Universal Robots PolyScope program: _adminCG-AssembleCLidToD.urp

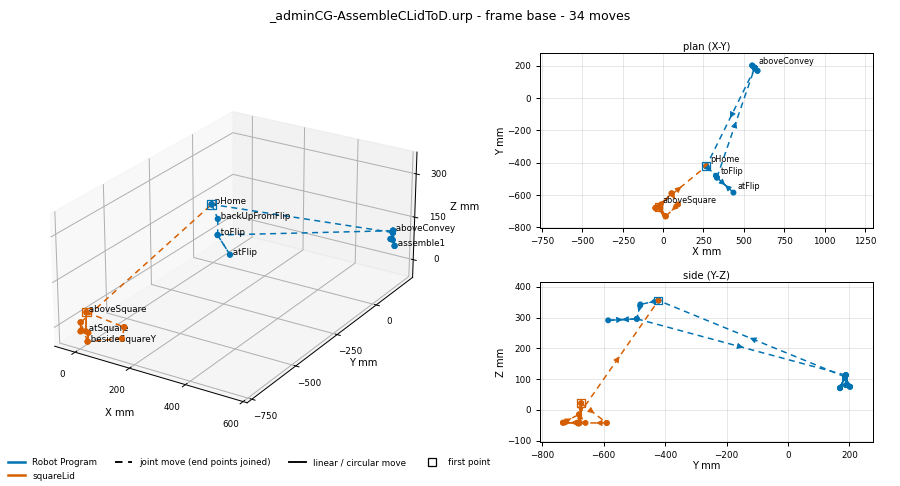
[picture p0: tool path of _adminCG-AssembleCLidToD.urp in frame base, 34 of 35 moves have a stored position in this frame; points joined in program order, loops and branches not executed]
Program _adminCG-AssembleCLidToD (installation=admin directory=/programs/WED_9AM createdIn=3.15.8.106339 lastSavedIn=3.15.8.106339 robotSerialNumber=2015350924)
Calibrated DH parameters: a=[0, -0.425, -0.39225, 0, 0, 0]; d=[0.089159, 0, 0, 0.10915, 0.09465, 0.0823]; alpha=[1.570796, 0, 0, 1.570796, -1.570796, 0]; deltaTheta=[0, 0, 0, 0, 0, 0]
Robot Program (runOnlyOnce=true)
  Set DigitalOutput pin=digital_out[0]; digitalValue=0
  MoveJ speed 60 deg/s, acceleration 80 deg/s^2 (useActiveTCP=true)
    Waypoint pHome: TCP in base x=267.157 y=-421.439 z=355.893 mm, rx=1.1139 ry=1.106 rz=0.0052 rad; joints [-44.996, -89.999, -89.997, -90.001, 90.007, 0.005] deg; flange x=267.148 y=-421.443 z=431.893 mm, rx=-1.2022 ry=2.9023 rz=0 rad
    Waypoint backUpFromFlip: TCP in base x=326.754 y=-480.276 z=343.158 mm, rx=1.1302 ry=1.1244 rz=-0.0012 rad; joints [-44.863, -101.867, -78.33, -91.204, 89.722, 0.314] deg; flange x=328.332 y=-481.325 z=419.134 mm, rx=1.1925 ry=-2.8912 rz=-0.0323 rad
  MoveJ speed 60 deg/s, acceleration 80 deg/s^2 (useActiveTCP=true)
    Call _adminLinearIndex4
    Waypoint toFlip: TCP in base x=333.102 y=-491.704 z=296.298 mm, rx=-1.5769 ry=1.6129 rz=-2.1772 rad; joints [-45.149, -123.398, -107.093, -41.475, -89.463, -0.24] deg; flange x=331.768 y=-489.353 z=220.346 mm, rx=0.0362 ry=0.0046 rz=0.7784 rad
    Waypoint atFlip: TCP in base x=435.484 y=-584.937 z=291.512 mm, rx=1.5199 ry=-1.5359 rz=2.2678 rad; joints [-44.833, -139.316, -77.941, -49.924, -90.495, -0.843] deg; flange x=437.672 y=-588.039 z=215.607 mm, rx=-0.0499 ry=-0.0116 rz=0.7732 rad
    Set DigitalOutput pin=digital_out[0]; digitalValue=1
    Wait Sleep waitTime=1
    Set DigitalOutput pin=digital_out[2]; digitalValue=0
    Wait Sleep waitTime=1
    Waypoint toFlip: TCP in base x=333.102 y=-491.704 z=296.298 mm, rx=-1.5769 ry=1.6129 rz=-2.1772 rad; joints [-45.149, -123.398, -107.093, -41.475, -89.463, -0.24] deg; flange x=331.768 y=-489.353 z=220.346 mm, rx=0.0362 ry=0.0046 rz=0.7784 rad
    Call _adminLinearIndex2
    Call squareLid
  MoveJ speed 60 deg/s, acceleration 80 deg/s^2 (useActiveTCP=true)
    Call _adminLinearIndex1
    Waypoint aboveConvey: TCP in base x=567.181 y=188.05 z=113.063 mm, rx=1.0282 ry=1.0751 rz=-0.0229 rad; joints [30.268, -112.359, -99.942, -58.865, 84.81, 74.946] deg; flange x=565.046 y=194.763 z=188.736 mm, rx=1.2073 ry=-2.8879 rz=0.1448 rad
    Waypoint rotateAbove: TCP in base x=567.194 y=188.064 z=113.07 mm, rx=1.5788 ry=-1.6466 rz=-2.1023 rad; joints [30.269, -112.36, -99.938, -58.868, 84.807, 254.946] deg; flange x=565.057 y=194.781 z=188.743 mm, rx=2.8131 ry=1.1761 rz=-0.0125 rad
    Waypoint atBody: TCP in base x=567.179 y=188.066 z=80.552 mm, rx=1.5785 ry=-1.6465 rz=-2.1025 rad; joints [30.268, -114.89, -101.837, -54.448, 84.816, 254.947] deg; flange x=565.059 y=194.78 z=156.225 mm, rx=2.8132 ry=1.1761 rz=-0.0127 rad
    Wait Sleep waitTime=1
    Set DigitalOutput pin=digital_out[0]; digitalValue=0
    Wait Sleep waitTime=1
    Waypoint rotateAbove: TCP in base x=567.194 y=188.064 z=113.07 mm, rx=1.5788 ry=-1.6466 rz=-2.1023 rad; joints [30.269, -112.36, -99.938, -58.868, 84.807, 254.946] deg; flange x=565.057 y=194.781 z=188.743 mm, rx=2.8131 ry=1.1761 rz=-0.0125 rad
    Waypoint aboveConvey: TCP in base x=567.181 y=188.05 z=113.063 mm, rx=1.0282 ry=1.0751 rz=-0.0229 rad; joints [30.268, -112.359, -99.942, -58.865, 84.81, 74.946] deg; flange x=565.046 y=194.763 z=188.736 mm, rx=1.2073 ry=-2.8879 rz=0.1448 rad
    Set DigitalOutput pin=digital_out[0]; digitalValue=1
    Waypoint abovePress: TCP in base x=568.039 y=185.31 z=107.717 mm, rx=1.0319 ry=1.117 rz=-0.0467 rad; joints [29.644, -113.286, -98.834, -61.278, 86.104, 74.264] deg; flange x=569.391 y=192.021 z=183.408 mm, rx=1.1944 ry=-2.8486 rz=0.1154 rad
  If force()≤65 (checkContinuously=true)
    MoveL speed 50 mm/s, acceleration 100 mm/s^2 (useActiveTCP=true) feature=Base
      Waypoint assemble1: TCP in base x=584.239 y=169.152 z=70.781 mm, rx=1.0609 ry=1.0742 rz=-0.0387 rad; joints [27.519, -116.934, -100.349, -53.785, 86.094, 73.63] deg; flange x=583.102 y=174.396 z=146.592 mm, rx=1.1698 ry=-2.9008 rz=0.109 rad
  MoveJ speed 60 deg/s, acceleration 80 deg/s^2 (useActiveTCP=true)
    Waypoint abovePress: TCP in base x=568.039 y=185.31 z=107.717 mm, rx=1.0319 ry=1.117 rz=-0.0467 rad; joints [29.644, -113.286, -98.834, -61.278, 86.104, 74.264] deg; flange x=569.391 y=192.021 z=183.408 mm, rx=1.1944 ry=-2.8486 rz=0.1154 rad
  If force()≤65 (checkContinuously=true)
    MoveL speed 50 mm/s, acceleration 100 mm/s^2 (useActiveTCP=true) feature=Base
      Waypoint assemble2: TCP in base x=551.811 y=201.79 z=75.225 mm, rx=1.0098 ry=1.1381 rz=-0.0159 rad; joints [31.851, -114.685, -102.439, -56.33, 86.144, 74.216] deg; flange x=552.994 y=208.542 z=150.915 mm, rx=1.2503 ry=-2.8248 rz=0.116 rad
  MoveJ speed 60 deg/s, acceleration 80 deg/s^2 (useActiveTCP=true)
    Waypoint abovePress: TCP in base x=568.039 y=185.31 z=107.717 mm, rx=1.0319 ry=1.117 rz=-0.0467 rad; joints [29.644, -113.286, -98.834, -61.278, 86.104, 74.264] deg; flange x=569.391 y=192.021 z=183.408 mm, rx=1.1944 ry=-2.8486 rz=0.1154 rad
  If force()≤65 (checkContinuously=true)
    MoveL speed 50 mm/s, acceleration 100 mm/s^2 (useActiveTCP=true) feature=Base
      Waypoint assemble1: TCP in base x=584.239 y=169.152 z=70.781 mm, rx=1.0609 ry=1.0742 rz=-0.0387 rad; joints [27.519, -116.934, -100.349, -53.785, 86.094, 73.63] deg; flange x=583.102 y=174.396 z=146.592 mm, rx=1.1698 ry=-2.9008 rz=0.109 rad
  MoveJ speed 60 deg/s, acceleration 80 deg/s^2 (useActiveTCP=true)
    Waypoint abovePress: TCP in base x=568.039 y=185.31 z=107.717 mm, rx=1.0319 ry=1.117 rz=-0.0467 rad; joints [29.644, -113.286, -98.834, -61.278, 86.104, 74.264] deg; flange x=569.391 y=192.021 z=183.408 mm, rx=1.1944 ry=-2.8486 rz=0.1154 rad
  If force()≤65 (checkContinuously=true)
    MoveL speed 50 mm/s, acceleration 100 mm/s^2 (useActiveTCP=true) feature=Base
      Waypoint assemble2: TCP in base x=551.811 y=201.79 z=75.225 mm, rx=1.0098 ry=1.1381 rz=-0.0159 rad; joints [31.851, -114.685, -102.439, -56.33, 86.144, 74.216] deg; flange x=552.994 y=208.542 z=150.915 mm, rx=1.2503 ry=-2.8248 rz=0.116 rad
  MoveJ speed 60 deg/s, acceleration 80 deg/s^2 (useActiveTCP=true)
    Waypoint abovePress: TCP in base x=568.039 y=185.31 z=107.717 mm, rx=1.0319 ry=1.117 rz=-0.0467 rad; joints [29.644, -113.286, -98.834, -61.278, 86.104, 74.264] deg; flange x=569.391 y=192.021 z=183.408 mm, rx=1.1944 ry=-2.8486 rz=0.1154 rad
    Waypoint pHome: TCP in base x=267.157 y=-421.439 z=355.893 mm, rx=1.1139 ry=1.106 rz=0.0052 rad; joints [-44.996, -89.999, -89.997, -90.001, 90.007, 0.005] deg; flange x=267.148 y=-421.443 z=431.893 mm, rx=-1.2022 ry=2.9023 rz=0 rad
SubProgram -> _adminLinearIndex1
SubProgram -> _adminLinearIndex4
SubProgram -> squareLid
SubProgram _adminLinearIndex3 (keepSynchronizedWithDisk=false) programFile=/programs/me345_admin/_adminLinearIndex3.urp
  Folder Move_linear_slide_Index1
    var_1 := False
    Loop While (checkContinuously=false) expression=var_1≟ False
      var_1 := socket_open("10.241.34.52",4001)
    var_3 := 1
    Send := "s r0x24 21"
    Script: socket_send_string(Send)
    Script: socket_send_byte(13)
    Send_Reply := socket_read_string()
    Send := "s r0xca 103936"
    Script: socket_send_string(Send)
    Script: socket_send_byte(13)
    Send_Reply := socket_read_string()
    Send := "t 1"
    Script: socket_send_string(Send)
    Script: socket_send_byte(13)
    Send_Reply := socket_read_string()
    Loop While (checkContinuously=false) expression=var_3≠0
      Send := "g r0xA0"
      Script: socket_send_string(Send)
      Script: socket_send_byte(13)
      var_3 := socket_get_var("v")
      Wait Sleep waitTime=0.1
    Script: socket_close()
    Script: sync()
SubProgram -> _adminLinearIndex2
SubProgram _adminLinearIndex5 (keepSynchronizedWithDisk=false) programFile=/programs/me345_admin/_adminLinearIndex5.urp
  Folder Move_linear_slide_Index5
    var_1 := False
    Loop While (checkContinuously=false) expression=var_1≟ False
      var_1 := socket_open("10.241.34.52",4001)
    var_3 := 1
    Send := "s r0x24 21"
    Script: socket_send_string(Send)
    Script: socket_send_byte(13)
    Send_Reply := socket_read_string()
    Send := "s r0xca 190000"
    Script: socket_send_string(Send)
    Script: socket_send_byte(13)
    Send_Reply := socket_read_string()
    Send := "t 1"
    Script: socket_send_string(Send)
    Script: socket_send_byte(13)
    Send_Reply := socket_read_string()
    Loop While (checkContinuously=false) expression=var_3≠0
      Send := "g r0xA0"
      Script: socket_send_string(Send)
      Script: socket_send_byte(13)
      var_3 := socket_get_var("v")
      Wait Sleep waitTime=0.1
    Script: socket_close()
    Script: sync()
SubProgram _adminLinearIndex4 (keepSynchronizedWithDisk=false) programFile=/programs/me345_admin/_adminLinearIndex4.urp
  Folder Move_linear_slide_Index4
    var_1 := False
    Loop While (checkContinuously=false) expression=var_1≟ False
      var_1 := socket_open("10.241.34.52",4001)
    var_3 := 1
    Send := "s r0x24 21"
    Script: socket_send_string(Send)
    Script: socket_send_byte(13)
    Send_Reply := socket_read_string()
    Send := "s r0xca 169167"
    Script: socket_send_string(Send)
    Script: socket_send_byte(13)
    Send_Reply := socket_read_string()
    Send := "t 1"
    Script: socket_send_string(Send)
    Script: socket_send_byte(13)
    Send_Reply := socket_read_string()
    Loop While (checkContinuously=false) expression=var_3≠0
      Send := "g r0xA0"
      Script: socket_send_string(Send)
      Script: socket_send_byte(13)
      var_3 := socket_get_var("v")
      Wait Sleep waitTime=0.1
    Script: socket_close()
    Script: sync()
SubProgram _adminLinearIndex2 (keepSynchronizedWithDisk=false) programFile=/programs/me345_admin/_adminLinearIndex2.urp
  Folder Move_linear_slide_Index2
    var_1 := False
    Loop While (checkContinuously=false) expression=var_1≟ False
      var_1 := socket_open("10.241.34.52",4001)
    var_3 := 1
    Send := "s r0x24 21"
    Script: socket_send_string(Send)
    Script: socket_send_byte(13)
    Send_Reply := socket_read_string()
    Send := "s r0xca 51968"
    Script: socket_send_string(Send)
    Script: socket_send_byte(13)
    Send_Reply := socket_read_string()
    Send := "t 1"
    Script: socket_send_string(Send)
    Script: socket_send_byte(13)
    Send_Reply := socket_read_string()
    Loop While (checkContinuously=false) expression=var_3≠0
      Send := "g r0xA0"
      Script: socket_send_string(Send)
      Script: socket_send_byte(13)
      var_3 := socket_get_var("v")
      Wait Sleep waitTime=0.1
    Script: socket_close()
    Script: sync()
SubProgram squareLid (keepSynchronizedWithDisk=false) programFile=/programs/WED_9AM/squareLid.urp
  MoveJ speed 180 deg/s, acceleration 100 deg/s^2 (useActiveTCP=true)
    Waypoint aboveSquare: TCP in base x=-28.511 y=-672.755 z=21.747 mm, rx=1.7065 ry=-0.0121 rz=-1.2064 rad; joints [-83.109, -128.084, -90.371, -51.361, 90.044, 52.13] deg; flange x=-28.598 y=-672.52 z=97.746 mm, rx=1.2074 ry=2.8979 rz=-0.0038 rad
  MoveL speed 250 mm/s, acceleration 1200 mm/s^2 (useActiveTCP=true) feature=Base
    Waypoint atSquare: TCP in base x=-30.006 y=-677.246 z=-41.376 mm, rx=1.7064 ry=-0.0122 rz=-1.2062 rad; joints [-83.283, -134.212, -90.751, -44.844, 90.048, 51.953] deg; flange x=-30.099 y=-676.998 z=34.624 mm, rx=1.2073 ry=2.8978 rz=-0.004 rad
    Set DigitalOutput pin=digital_out[0]; digitalValue=0
    Wait Sleep waitTime=0.5
    Waypoint aboveSquare: TCP in base x=-28.511 y=-672.755 z=21.747 mm, rx=1.7065 ry=-0.0121 rz=-1.2064 rad; joints [-83.109, -128.084, -90.371, -51.361, 90.044, 52.13] deg; flange x=-28.598 y=-672.52 z=97.746 mm, rx=1.2074 ry=2.8979 rz=-0.0038 rad
    Set DigitalOutput pin=digital_out[0]; digitalValue=1
  MoveJ speed 60 deg/s, acceleration 80 deg/s^2 (useActiveTCP=true)
    Waypoint besideSquareX: TCP in base x=52.617 y=-589.571 z=-42.423 mm, rx=1.7065 ry=-0.0117 rz=-1.2076 rad; joints [-74.267, -126.531, -106.897, -36.426, 89.974, 61.001] deg; flange x=52.598 y=-589.375 z=33.577 mm, rx=1.2085 ry=2.8985 rz=-0.0036 rad
  MoveL speed 35 mm/s, acceleration 35 mm/s^2 (useActiveTCP=true) feature=Base
    If force()≤40 (checkContinuously=true)
      Waypoint atSquareX_1 (Relative): relativeFromPosition TCP in base x=50.865 y=-591.008 z=-41.515 mm, rx=1.7022 ry=-0.008 rz=-1.2089 rad; joints [-74.266, -126.532, -106.898, -36.426, 89.971, 60.977] deg; TCP in base x=-28.314 y=-672.475 z=-41.562 mm, rx=1.7067 ry=-0.0121 rz=-1.2064 rad; joints [-83.089, -133.766, -91.707, -44.351, 90.046, 52.151] deg; flange x=-28.404 y=-672.249 z=34.438 mm, rx=1.2075 ry=2.8979 rz=-0.0036 rad
    Wait Sleep waitTime=0.5
  MoveJ speed 60 deg/s, acceleration 80 deg/s^2 (useActiveTCP=true)
    Waypoint besideSquareX: TCP in base x=52.617 y=-589.571 z=-42.423 mm, rx=1.7065 ry=-0.0117 rz=-1.2076 rad; joints [-74.267, -126.531, -106.897, -36.426, 89.974, 61.001] deg; flange x=52.598 y=-589.375 z=33.577 mm, rx=1.2085 ry=2.8985 rz=-0.0036 rad
    Waypoint linkingMove: motionParameters(blendRadius=0.01); TCP in base x=92.406 y=-658.703 z=-42.29 mm, rx=1.7071 ry=-0.0114 rz=-1.2067 rad; joints [-72.572, -133.085, -93.255, -43.522, 90.01, 62.663] deg; flange x=92.339 y=-658.532 z=33.709 mm, rx=1.2075 ry=2.8984 rz=-0.0027 rad
    Waypoint besideSquareY: TCP in base x=16.11 y=-732.019 z=-41.564 mm, rx=1.7069 ry=-0.0118 rz=-1.2058 rad; joints [-80.178, -139.758, -79.322, -50.745, 90.056, 55.034] deg; flange x=15.998 y=-731.803 z=34.435 mm, rx=1.2067 ry=2.8979 rz=-0.0032 rad
  MoveL speed 35 mm/s, acceleration 35 mm/s^2 (useActiveTCP=true) feature=Base
    If force()≤40 (checkContinuously=true)
      Waypoint atSquareY_1: TCP in base x=-16.892 y=-681.869 z=-41.456 mm, rx=1.7062 ry=-0.0123 rz=-1.2065 rad; joints [-82.218, -134.623, -89.92, -45.26, 90.031, 53.025] deg; flange x=-16.969 y=-681.614 z=34.543 mm, rx=1.2075 ry=2.8978 rz=-0.0043 rad
    Wait Sleep waitTime=0.5
  MoveJ speed 60 deg/s, acceleration 80 deg/s^2 (useActiveTCP=true)
    Waypoint besideSquareY: TCP in base x=16.11 y=-732.019 z=-41.564 mm, rx=1.7069 ry=-0.0118 rz=-1.2058 rad; joints [-80.178, -139.758, -79.322, -50.745, 90.056, 55.034] deg; flange x=15.998 y=-731.803 z=34.435 mm, rx=1.2067 ry=2.8979 rz=-0.0032 rad
    Waypoint aboveSquareNew: TCP in base x=-46.625 y=-679.478 z=-14.514 mm, rx=1.7065 ry=-0.012 rz=-1.2064 rad; joints [-84.714, -132.04, -89.733, -48.043, 90.045, 50.52] deg; flange x=-46.706 y=-679.241 z=61.486 mm, rx=1.2073 ry=2.898 rz=-0.0039 rad
    Set DigitalOutput pin=digital_out[0]; digitalValue=0
    Wait Sleep waitTime=1
  MoveL speed 250 mm/s, acceleration 1200 mm/s^2 (useActiveTCP=true) feature=Base
    Waypoint atSquareNew: TCP in base x=-46.857 y=-681.738 z=-44.514 mm, rx=1.7064 ry=-0.0116 rz=-1.2062 rad; joints [-84.751, -135.038, -89.679, -45.105, 90.044, 50.462] deg; flange x=-46.937 y=-681.507 z=31.486 mm, rx=1.2068 ry=2.8982 rz=-0.0038 rad
    Set DigitalOutput pin=digital_out[0]; digitalValue=1
    Wait Sleep waitTime=1
    Waypoint easeout: TCP in base x=-46.631 y=-679.453 z=-43.525 mm, rx=1.7066 ry=-0.0121 rz=-1.2065 rad; joints [-84.715, -134.722, -90.131, -44.972, 90.046, 50.528] deg; flange x=-46.714 y=-679.227 z=32.475 mm, rx=1.2076 ry=2.8979 rz=-0.0037 rad
    Waypoint aboveSquareNew: TCP in base x=-46.625 y=-679.478 z=-14.514 mm, rx=1.7065 ry=-0.012 rz=-1.2064 rad; joints [-84.714, -132.04, -89.733, -48.043, 90.045, 50.52] deg; flange x=-46.706 y=-679.241 z=61.486 mm, rx=1.2073 ry=2.898 rz=-0.0039 rad
  MoveJ speed 60 deg/s, acceleration 80 deg/s^2 (useActiveTCP=true)
    Waypoint pHome_1: TCP in base x=267.157 y=-421.439 z=355.893 mm, rx=1.1139 ry=1.106 rz=0.0052 rad; joints [-44.996, -89.999, -89.997, -90.001, 90.007, 0.005] deg; flange x=267.148 y=-421.443 z=431.893 mm, rx=-1.2022 ry=2.9023 rz=0 rad
SubProgram _adminLinearIndex1 (keepSynchronizedWithDisk=false) programFile=/programs/me345_admin/_adminLinearIndex1.urp
  Folder Move_linear_slide_Index1
    var_1 := False
    Loop While (checkContinuously=false) expression=var_1≟ False
      var_1 := socket_open("10.241.34.52",4001)
    var_3 := 1
    Send := "s r0x24 21"
    Script: socket_send_string(Send)
    Script: socket_send_byte(13)
    Send_Reply := socket_read_string()
    Send := "s r0xca 0"
    Script: socket_send_string(Send)
    Script: socket_send_byte(13)
    Send_Reply := socket_read_string()
    Send := "t 1"
    Script: socket_send_string(Send)
    Script: socket_send_byte(13)
    Send_Reply := socket_read_string()
    Loop While (checkContinuously=false) expression=var_3≠0
      Send := "g r0xA0"
      Script: socket_send_string(Send)
      Script: socket_send_byte(13)
      var_3 := socket_get_var("v")
      Wait Sleep waitTime=0.1
    Script: socket_close()
    Script: sync()
